(* IEC 61131-3 sources: AXOpen/src/core/ctrl/src, 4 files *)

(* ---- IxObject.st ---- *)
NAMESPACE ix.framework.core

    FUNCTION IsNullContext : BOOL
        VAR_INPUT
            Context : IIxContext;
        END_VAR
        IF Context = NULL THEN
            IsNullContext := TRUE;
        ELSIF Context.CreateIdentity() = ULINT#0 THEN
            IsNullContext := TRUE;
        ELSE
            IsNullContext := FALSE;
        END_IF;
    END_FUNCTION

    ///<summary>
    /// Provides an empty context for uninitialized objects.
    ///</summary>
    CLASS PUBLIC _NULL_CONTEXT IMPLEMENTS IIxContext
        METHOD PUBLIC CreateIdentity : ULINT CreateIdentity := ULINT#0; END_METHOD
        METHOD PUBLIC OpenCycleCount : ULINT OpenCycleCount := ULINT#0; END_METHOD
    END_CLASS

    ///<summary>
    /// Provides an empty object for uninitialized objects.
    ///</summary>
    CLASS PUBLIC _NULL_OBJECT IMPLEMENTS IIxObject
        VAR PRIVATE
            NULL_CONTEXT : _NULL_CONTEXT;
        END_VAR
        METHOD PUBLIC GetIdentity : ULINT
            GetIdentity := ULINT#0;
        END_METHOD
        METHOD PUBLIC GetContext : IIxContext
            GetContext := NULL_CONTEXT;
        END_METHOD
    END_CLASS

    ///<summary>
    /// Provides base class for all classes of `ix.framework`.
    ///</summary>
    CLASS PUBLIC IxObject IMPLEMENTS IIxObject
        VAR PUBLIC
            {#ix-attr:[CompilerOmits("POCO")]}
            {#ix-attr:[ReadOnly()]}
            Identity   : ULINT := ULINT#0;
        END_VAR

        VAR PRIVATE
            _parent     : IIxObject;
            _context    : IIxContext;
        END_VAR

        VAR PRIVATE
            NULL_CONTEXT : _NULL_CONTEXT;
            NULL_OBJECT : _NULL_OBJECT;
        END_VAR

        ///<summary>
        /// Gets unique identity of this object in given context.
        ///</summary>
        METHOD PUBLIC GetIdentity : ULINT
            GetIdentity := Identity;
        END_METHOD

        ///<summary>
        /// Gets context in which this object was initialized.
        ///</summary>
        METHOD PUBLIC GetContext : IIxContext
            IF(_context <> NULL) THEN
                GetContext := _context;
            ELSE
                GetContext := NULL_CONTEXT;
            END_IF;
        END_METHOD

        ///<summary>
        /// Gets parent in which this object was initialized.
        ///</summary>
        METHOD PUBLIC GetParent : IIxObject
            IF(_context <> NULL) THEN
                GetParent := _parent;
            ELSE
                GetParent := NULL_OBJECT;
            END_IF;
        END_METHOD

        ///<summary>
        /// Initializes this object associating it given parent.
        /// This method should be called only once upon the program start.
        /// Any subsequent call are ignored.
        ///</summary>
        METHOD PUBLIC Initialize
            VAR_INPUT
                parent : IIxObject;
            END_VAR

            IF(Identity = ULINT#0 AND parent <> NULL) THEN
                _context    := parent.GetContext();
                Identity   := _context.CreateIdentity();
                _parent     := parent;
                RETURN;
            END_IF;

        END_METHOD

        ///<summary>
        /// Initializes this object associating it given context.
        /// This method should be called only once upon the program start.
        /// Any subsequent call are ignored.
        ///</summary>
        METHOD PUBLIC Initialize
            VAR_INPUT
                context : IIxContext;
            END_VAR

            IF(Identity = ULINT#0 AND context <> NULL) THEN
                _context    := context;
                Identity   := _context.CreateIdentity();
            END_IF;

        END_METHOD
    END_CLASS
END_NAMESPACE

(* ---- Object.st ---- *)
NAMESPACE ix.framework.core

    FUNCTION IsNullContext : BOOL
        VAR_INPUT
            Context : IContext;
        END_VAR
        IF Context = NULL THEN
            IsNullContext := TRUE;
        ELSIF Context.CreateIdentity() = ULINT#0 THEN
            IsNullContext := TRUE;
        ELSE
            IsNullContext := FALSE;
        END_IF;
    END_FUNCTION

    ///<summary>
    /// Provides an empty context for uninitialized objects.
    ///</summary>
    CLASS PUBLIC _NULL_CONTEXT IMPLEMENTS IContext
        METHOD PUBLIC CreateIdentity : ULINT CreateIdentity := ULINT#0; END_METHOD
        METHOD PUBLIC OpenCycleCount : ULINT OpenCycleCount := ULINT#0; END_METHOD
    END_CLASS

    ///<summary>
    /// Provides base class for all classes of `ix.framework`.
    ///</summary>
    CLASS PUBLIC Object IMPLEMENTS IObject
        VAR PRIVATE
            _identity   : ULINT := ULINT#0;
            _parent     : IObject;
            _context    : IContext;
        END_VAR

        VAR PRIVATE
            NULL_CONTEXT : _NULL_CONTEXT;
        END_VAR

        ///<summary>
        /// Gets unique identity of this object in given context.
        ///</summary>
        METHOD PUBLIC GetIdentity : ULINT
            GetIdentity := _identity;
        END_METHOD

        ///<summary>
        /// Gets context in which this object was initialized.
        ///</summary>
        METHOD PUBLIC GetContext : IContext
            IF(_context <> NULL) THEN
                GetContext := _context;
            ELSE
                GetContext := NULL_CONTEXT;
            END_IF;
        END_METHOD

        ///<summary>
        /// Initializes this object associating it given parent.
        /// This method should be called only once upon the program start.
        /// Any subsequent call are ignored.
        ///</summary>
        METHOD PUBLIC Initialize
            VAR_INPUT
                parent : IObject;
            END_VAR

            IF(_identity = ULINT#0 AND parent <> NULL) THEN
                _context    := parent.GetContext();
                _identity   := _context.CreateIdentity();
                _parent     := parent;
                RETURN;
            END_IF;

        END_METHOD

        ///<summary>
        /// Initializes this object associating it given context.
        /// This method should be called only once upon the program start.
        /// Any subsequent call are ignored.
        ///</summary>
        METHOD PUBLIC Initialize
            VAR_INPUT
                context : IContext;
            END_VAR

            IF(_identity = ULINT#0 AND context <> NULL) THEN
                _context    := context;
                _identity   := _context.CreateIdentity();
            END_IF;

        END_METHOD
    END_CLASS
END_NAMESPACE

(* ---- Context.st ---- *)
NAMESPACE ix.framework.core
    ///<summary>
    /// Provides base for contextualized entry of `ix.framework` application.
    /// This class is abstract and must be inherited.
    ///</summary>
    CLASS PUBLIC ABSTRACT Context IMPLEMENTS IContext
        VAR PRIVATE
            _openCounter : ULINT;
            _closeCounter : ULINT;
            _identityCounter : ULINT;
        END_VAR

        ///<summary>
        /// The entry point for the context. The call tree of the context start here and all the logic of given context
        /// must be placed here.
        /// This method must be overridden in derived class.
        ///</summary>
        METHOD PROTECTED ABSTRACT Main END_METHOD

        METHOD PRIVATE Open : ULINT
            _openCounter := _openCounter + ULINT#1;
        END_METHOD

        METHOD PRIVATE Close : ULINT
            _closeCounter := _closeCounter + ULINT#1;
        END_METHOD

        ///<summary>
        /// Executes the cycle of this context. This method must be called cyclically in a PLC task.
        ///</summary>
        METHOD PUBLIC Execute
            THIS.Open();
            THIS.Main();
            THIS.Close();
        END_METHOD

        ///<summary>
        /// Gets the value of current context cycle counter.
        ///</summary>
        METHOD PUBLIC OpenCycleCount : ULINT
            OpenCycleCount := _openCounter;
        END_METHOD

        METHOD PUBLIC ClosedCycleCount : ULINT
            ClosedCycleCount := _closeCounter;
        END_METHOD

        METHOD PUBLIC CreateIdentity : ULINT
            _identityCounter := _identityCounter + ULINT#1;
            CreateIdentity := _identityCounter;
        END_METHOD

        METHOD PUBLIC PeekIdentity : ULINT
            PeekIdentity := _identityCounter;
        END_METHOD

    END_CLASS
END_NAMESPACE

(* ---- IxContext.st ---- *)
NAMESPACE ix.framework.core
    ///<summary>
    /// Provides base for contextualized entry of `ix.framework` application.
    /// This class is abstract and must be inherited.
    ///</summary>
    CLASS PUBLIC ABSTRACT IxContext IMPLEMENTS IIxContext
        VAR PRIVATE
            _openCounter : ULINT;
            _closeCounter : ULINT;
            _identityCounter : ULINT;
        END_VAR

        ///<summary>
        /// The entry point for the context. The call tree of the context start here and all the logic of given context
        /// must be placed here.
        /// This method must be overridden in derived class.
        ///</summary>
        METHOD PROTECTED ABSTRACT Main END_METHOD

        METHOD PRIVATE Open : ULINT
            _openCounter := _openCounter + ULINT#1;
        END_METHOD

        METHOD PRIVATE Close : ULINT
            _closeCounter := _closeCounter + ULINT#1;
        END_METHOD

        ///<summary>
        /// Executes the cycle of this context. This method must be called cyclically in a PLC task.
        ///</summary>
        METHOD PUBLIC Execute
            THIS.Open();
            THIS.Main();
            THIS.Close();
        END_METHOD

        ///<summary>
        /// Gets the value of current context cycle counter.
        ///</summary>
        METHOD PUBLIC OpenCycleCount : ULINT
            OpenCycleCount := _openCounter;
        END_METHOD

        METHOD PUBLIC ClosedCycleCount : ULINT
            ClosedCycleCount := _closeCounter;
        END_METHOD

        METHOD PUBLIC CreateIdentity : ULINT
            _identityCounter := _identityCounter + ULINT#1;
            CreateIdentity := _identityCounter;
        END_METHOD

        METHOD PUBLIC PeekIdentity : ULINT
            PeekIdentity := _identityCounter;
        END_METHOD

    END_CLASS
END_NAMESPACE
